// TwinCAT 3 PLC project lev_fsm
// ProgramVersion: 3.1.4023.0
// libraries:
//   Tc2_SerialCom, * (Beckhoff Automation GmbH)
//   Tc2_Standard, * (Beckhoff Automation GmbH)
//   Tc2_System, * (Beckhoff Automation GmbH)
//   Tc2_Utilities, * (Beckhoff Automation GmbH)
//   Tc3_Module, * (Beckhoff Automation GmbH)
// project tree:
//   DUTs/ E_FsmError.TcDUT, E_FsmState.TcDUT, mag_bus.TcDUT, ST_Event.TcDUT, sus_bus.TcDUT
//   / PlcTask.TcTTO
//   POUs/ getTrajectory.TcPOU (not stored), LevitationEqualizingController.TcPOU, MAIN.TcPOU, runIpcFsm.TcPOU (not stored)
//   POUs/outdated/ FiniteStateMachine.TcPOU (not stored), GenerateTrajectory.TcPOU, getFmagnetic.TcPOU, Trajectory.TcPOU (not stored), UpdateEventTimestampWithSystemTime.TcPOU (not stored)

CONFIGURATION lev_fsm
    RESOURCE PLC ON TwinCAT3
        TASK PlcTask(INTERVAL := T#10ms, PRIORITY := 6);
        PROGRAM MAIN WITH PlcTask : MAIN;
    END_RESOURCE
END_CONFIGURATION

// ---- DUTs/E_FsmError.TcDUT
{attribute 'qualified_only'}
{attribute 'strict'}
{attribute 'to_string'}
TYPE E_FsmError :
(
	NO_ERR		  := 0,
	INIT_ERR      := 1,
	STAT_ERR      := 2,
	STAT_TR_ERR   := 3,
	NOM_LEV_ERR   := 4,
	INTER_TR_ERR  := 5,
	END_TR_ERR    := 6
);
END_TYPE

// ---- DUTs/E_FsmState.TcDUT
{attribute 'qualified_only'}
{attribute 'strict'}
{attribute 'to_string'}
TYPE E_FsmState :
(
	ERR       := 0,
	INIT      := 1,
	STAT      := 2, 
	STAT_TR   := 3,
	NOM_LEV   := 4,
	INTER_TR  := 5,
	END_TR 	  := 6
);
END_TYPE

// ---- DUTs/mag_bus.TcDUT
TYPE mag_bus:
    STRUCT
        Fmat: ARRAY [0..143] OF LREAL;
        zmat: ARRAY [0..143] OF LREAL;
        invFmat: ARRAY [0..143] OF LREAL;
        F_grid: ARRAY [0..16383] OF LREAL;
        z_grid: ARRAY [0..16383] OF LREAL;
        i_grid: ARRAY [0..16383] OF LREAL;
    END_STRUCT
END_TYPE

// ---- DUTs/ST_Event.TcDUT
TYPE ST_Event :
STRUCT
	eEventType : E_TcEventClass;
	eEventSeverity : TcEventSeverity;
	nEventID : UDINT;
	sEventDescription : STRING(255);
	dtTimestamp : DATE_AND_TIME;
END_STRUCT
END_TYPE

// ---- DUTs/sus_bus.TcDUT
TYPE sus_bus:
    STRUCT
        zmax: LREAL;
        zcont: LREAL;
    END_STRUCT
END_TYPE

// ---- POUs/MAIN.TcPOU
PROGRAM MAIN

VAR CONSTANT
	tTIMER_TRESHOLD: TIME := T#10S;
END_VAR

VAR
	// LOGGING 
	fbOpenLogFile : FB_FileOpen := (sPathName:='.\logs\ipc.log', nMode:= FOPEN_MODEAPPEND OR FOPEN_MODETEXT);
    fbPutsLogFile : FB_FilePuts;		
	// Reference vector
	x_ref : ARRAY[1..3] OF REAL := [0.01, 0, 32.5]; // [z_nom, v_des, I_nom]
	z_nom : REAL := x_ref[1]; // Nominal air gap
	v_des : REAL := x_ref[2]; // Desired vertical velocity at nominal state
	I_nom: REAL := x_ref[3]; // Nominal current	
	eFsmState : E_FsmState := E_FsmState.INIT; // Finite State Machine State initialization
	eNextFsmState : E_FsmState := E_FsmState.INIT; // Next Finite State Machine State initialization
	stEvent : ST_Event; // Finite State Machine Event definition
	eFsmErrorStatus : E_FsmError; // Finite State Machine Error status
	
	fbTimer: TON := (PT:= tTIMER_TRESHOLD);
	bTimerStart: BOOL := TRUE;
	
	pz_nom : POINTER TO REAL := ADR(z_nom);
	rz_nom : REFERENCE TO REAL REF=z_nom;
	bRunOnlyOnce: BOOL := FALSE;
	nSizeOfLoggerMessage: UINT;
	sLoggerMessage: STRING(100) := 'Logging Finite State Machine State';
	tTime: TIME := T#0D0H0M0S0MS;
	
	// Levitation Equalizing Controller
	fSetpointValue : LREAL := 0; // Reference delta F = 0 N
	bReset : BOOL; // Reset flag for PID block
	fCtrlCycleTime : LREAL := 0.1; // Update cycle time of PID block
	fKp : LREAL := 1/1000;  // Proportional gain of PID block
	fTn : LREAL := 1/150; 
	fTv : LREAL := 0;
	fTd : LREAL := 0;
	fCtrlOutput : LREAL; // Output of PID block
	nErrorStatus : UINT; // Error status of levitation equalizing controller
	// Levitation equalizing controller function block initialization
	LevEqCtrl : LevitationEqualizingController(fSetpointValue := fSetpointValue,
											   bReset := bReset,
                                               fCtrlCycleTime := fCtrlCycleTime,
											   fKp := fKp,
											   fTn := fTn,
											   fTv := fTv,
											   fTd := fTd);
	fActualdF : LREAL; // Actual delta F = (F1 + F3) - (F2 + F4)
	fdz : ARRAY[1..4] OF LREAL;	// dz output vector of levitation equalizing controller
	// Forces
	fFmagFL : LREAL;
	fFmagFR : LREAL;
	fFmagBR : LREAL;
	fFmagBL : LREAL;
	// Test current, airgap and magnetic force
	fztest : LREAL;
	fItest : LREAL;
	fFmagtest : LREAL;
END_VAR

eFsmErrorStatus := runIpcFsm(eFsmState, eNextFsmState, fbTimer, bTimerStart);
fActualdF := (fFmagFL + fFmagBR) - (fFmagFR + fFmagBL);
LevEqCtrl(fActualdF := fActualdF, fdz => fdz, nErrorStatus => nErrorStatus);

fFmagtest := getFmagnetic(fItest,fztest);





(*
IF NOT bRunOnlyOnce THEN
	eNextFsmState := FiniteStateMachine(eArgFsmState := eFsmState);
	pz_nom^ := 0.015;
	x_ref := GenerateTrajectory(z_meas := 0.015, v_meas := 0.01, I_meas := 40);
	stEvent.sEventDescription := 'Start magnetic suspension';
	UpdateEventTimestampWithSystemTime(stEvent := stEvent);
	nSizeOfLoggerMessage := SIZEOF(sLoggerMessage);
	ADSLOGSTR(msgCtrlMask := ADSLOG_MSGTYPE_ERROR OR ADSLOG_MSGTYPE_LOG, 
		  msgFmtStr := sLoggerMessage,
		  strArg := '');
	bRunOnlyOnce := TRUE;
END_IF	 
*)

END_PROGRAM

// ---- POUs/LevitationEqualizingController.TcPOU
FUNCTION_BLOCK LevitationEqualizingController
VAR_INPUT
	// Actual delta F value
	fActualdF : LREAL;
END_VAR

VAR
	// PID function block	
	fbPID : FB_BasicPID;
	// PID parameters
	fSetpointValue : LREAL;
	bReset : BOOL;
	fCtrlCycleTime : LREAL;
	fKp : LREAL;
	fTn : LREAL;
	fTv : LREAL;
	fTd : LREAL;
	// PID outputs	
	fCtrlOutput : LREAL;
	// Saturation parameter
	fdzMax : LREAL := 0.001;
	fdzMin : LREAL := -0.001;
END_VAR
VAR_OUTPUT
	// dz output vector
	fdz : ARRAY[1..4] OF LREAL;
	nErrorStatus : UINT;
END_VAR

fbPID(fSetpointValue := fSetpointValue,
	  fActualValue := fActualdF,
	  bReset := bReset,
	  fCtrlCycleTime := fCtrlCycleTime,
	  fKp := fKp,
	  fTn := fTn,
	  fTv := fTv,
	  fTd := fTd,
	  fCtrlOutput => fCtrlOutput, nErrorStatus => nErrorStatus);
	  
// Update the dz output vector
fdz[1] := -1/7900*fCtrlOutput; // TO DO : change it to lookup table function F_inv(F)
fdz[2] := 1/7900*fCtrlOutput;
fdz[3] := -1/7900*fCtrlOutput;
fdz[4] := 1/7900*fCtrlOutput;	  

// Saturate the dz output vector
IF fdz[1] > fdzMax THEN
	fdz[1] := fdzMax;
ELSIF fdz[1] < fdzMin THEN
	fdz[1] := fdzMin;
END_IF

IF fdz[2] > fdzMax THEN
	fdz[2] := fdzMax;
ELSIF fdz[2] < fdzMin THEN
	fdz[2] := fdzMin;
END_IF

IF fdz[3] > fdzMax THEN
	fdz[3] := fdzMax;
ELSIF fdz[3] < fdzMin THEN
	fdz[3] := fdzMin;
END_IF

IF fdz[4] > fdzMax THEN
	fdz[4] := fdzMax;
ELSIF fdz[4] < fdzMin THEN
	fdz[4] := fdzMin;
END_IF

METHOD FB_init : BOOL
VAR_INPUT
	bInitRetains : BOOL; // if TRUE, the retain variables are initialized (warm start / cold start)
	bInCopyCode : BOOL;  // if TRUE, the instance afterwards gets moved into the copy code (online change)
	fSetpointValue : LREAL;
	bReset : BOOL;
	fCtrlCycleTime : LREAL;
	fKp : LREAL;
	fTn : LREAL;
	fTv : LREAL;
	fTd : LREAL;
END_VAR
THIS^.fSetpointValue := fSetpointValue;
THIS^.bReset := bReset;
THIS^.fCtrlCycleTime := fCtrlCycleTime;
THIS^.fKp := fKp;
THIS^.fTn := fTn;
THIS^.fTv := fTv;
THIS^.fTd := fTd;
END_METHOD

END_FUNCTION_BLOCK

// ---- POUs/outdated/getFmagnetic.TcPOU
FUNCTION getFmagnetic : LREAL
VAR_INPUT
    I: LREAL;
    z: LREAL;
END_VAR
VAR
    Fmag_tmp: LREAL;
    Fmag_tmp_0: LREAL;
    Fmag_tmp_1: LREAL;
    Fmag_tmp_2: LREAL;
    Fmag_tmp_3: LREAL;
    Fmag_tmp_4: LREAL;
END_VAR

(* MATLAB Function: '<Root>/getFmag' *)
(* MATLAB Function 'getFmag': '<S1>:1' *)
(* '<S1>:1:2' p00 =  -4.108e+05; *)
(* '<S1>:1:3' p10 =        3267; *)
(* '<S1>:1:4' p01 =   1.697e+05; *)
(* '<S1>:1:5' p20 =       61.45; *)
(* '<S1>:1:6' p11 =       -1147; *)
(* '<S1>:1:7' p02 =   -2.79e+04; *)
(* '<S1>:1:8' p30 =     -0.5002; *)
(* '<S1>:1:9' p21 =      -8.054; *)
(* '<S1>:1:10' p12 =       147.8; *)
(* '<S1>:1:11' p03 =        2282; *)
(* '<S1>:1:12' p40 =    -0.01962; *)
(* '<S1>:1:13' p31 =      0.1688; *)
(* '<S1>:1:14' p22 =      0.1559; *)
(* '<S1>:1:15' p13 =      -8.184; *)
(* '<S1>:1:16' p04 =      -92.92; *)
(* '<S1>:1:17' p50 =   0.0002649; *)
(* '<S1>:1:18' p41 =   -0.001089; *)
(* '<S1>:1:19' p32 =   -0.001289; *)
(* '<S1>:1:20' p23 =   -0.003046; *)
(* '<S1>:1:21' p14 =      0.1725; *)
(* '<S1>:1:22' p05 =       1.506; *)
(* '<S1>:1:23' Fmag = p00 + p10*I + p01*z + p20*I^2 + p11*I*z + p02*z^2 + p30*I^3 + p21*I^2*z + p12*I*z^2 + p03*z^3 + p40*I^4 + p31*I^3*z + p22*I^2*z^2 + p13*I*z^3 + p04*z^4 + p50*I^5 + p41*I^4*z + p32*I^3*z^2 + p23*I^2*z^3 + p14*I*z^4 + p05*z^5; *)
Fmag_tmp := EXPT(I, 3.0);
Fmag_tmp_0 := EXPT(z, 3.0);
Fmag_tmp_1 := EXPT(I, 4.0);
Fmag_tmp_2 := EXPT(z, 4.0);
Fmag_tmp_3 := I * I;
Fmag_tmp_4 := z * z;
getFmagnetic := ((((((((((((((((((((3267.0 * I) - 410800.0) + (169700.0 * z)) + (Fmag_tmp_3 * 61.45)) + ((-1147.0 * I) * z)) + (Fmag_tmp_4 * -27900.0)) + (-0.5002 * Fmag_tmp)) + ((Fmag_tmp_3 * -8.054) * z)) + ((147.8 * I) * Fmag_tmp_4)) + (2282.0 * Fmag_tmp_0)) + (-0.01962 * Fmag_tmp_1)) + ((0.1688 * Fmag_tmp) * z)) + ((Fmag_tmp_3 * 0.1559) * Fmag_tmp_4)) + ((-8.184 * I) * Fmag_tmp_0)) + (-92.92 * Fmag_tmp_2)) + (0.0002649 * EXPT(I, 5.0))) + ((-0.001089 * Fmag_tmp_1) * z)) + ((-0.001289 * Fmag_tmp) * Fmag_tmp_4)) + ((Fmag_tmp_3 * -0.003046) * Fmag_tmp_0)) + ((0.1725 * I) * Fmag_tmp_2)) + (1.506 * EXPT(z, 5.0));

END_FUNCTION

// ---- POUs/outdated/GenerateTrajectory.TcPOU
(*FUNCTION GenerateTrajectory :  ARRAY[1..3] OF REAL
VAR_INPUT
	z_meas : REAL;
	v_meas : REAL;
	I_meas : REAL;
END_VAR
VAR
END_VAR*)
(*
 *
 * File: trajectory_generator.st
 *
 * IEC 61131-3 Structured Text (ST) code generated for subsystem "trajectory_generator/getTrajectory"
 *
 * Model name                      : trajectory_generator
 * Model version                   : 3.24
 * Model creator                   : xiaomi
 * Model last modified by          : xiaomi
 * Model last modified on          : Tue Oct 25 16:42:44 2022
 * Model sample time               : 0.0005s
 * Subsystem name                  : trajectory_generator/getTrajectory
 * Subsystem sample time           : 0.1s
 * Simulink PLC Coder version      : 3.7 (R2022b) 13-May-2022
 * ST code generated on            : Tue Oct 25 16:44:27 2022
 *
 * Target IDE selection            : Beckhoff TwinCAT 3
 * Test Bench included             : No
 *
 *)
FUNCTION_BLOCK GenerateTrajectory
VAR_INPUT
    ssMethodType: SINT;
    t: LREAL;
    Tdes: LREAL;
    z0: LREAL;
    v0: LREAL;
    a0: LREAL;
    zdes: LREAL;
    vdes: LREAL;
    ades: LREAL;
    sus_params: sus_bus;
    mag_params: mag_bus;
END_VAR
VAR_OUTPUT
    zd: LREAL;
    vd: LREAL;
    ad: LREAL;
    id: LREAL;
END_VAR
VAR
    zd_prev_not_empty: BOOL;
    zd_prev: LREAL;
    vd_prev_not_empty: BOOL;
    vd_prev: LREAL;
    ad_prev_not_empty: BOOL;
    ad_prev: LREAL;
    id_prev: LREAL;
END_VAR
VAR_TEMP
    b2: LREAL;
    Fsus: LREAL;
    K: LREAL;
    zd_norm: LREAL;
    Fmag_norm: LREAL;
    A: ARRAY [0..8] OF LREAL;
    B: ARRAY [0..2] OF LREAL;
    r1: DINT;
    r2: DINT;
    r3: DINT;
    maxval: LREAL;
    a21: LREAL;
    rtemp: DINT;
    v: ARRAY [0..29] OF LREAL;
    b_v: ARRAY [0..15] OF LREAL;
    ry: LREAL;
    b_mid_i: DINT;
    x_idx_1: LREAL;
    x_idx_2: LREAL;
    x_idx_0: LREAL;
    u: DINT;
    b_u: DINT;
END_VAR

VAR CONSTANT
    SS_INITIALIZE: SINT := 0;
    SS_STEP: SINT := 1;
END_VAR

(*GenerateTrajectory[1] := z_meas/2;
GenerateTrajectory[2] := 0;
GenerateTrajectory[3] := I_meas/2;*)
CASE ssMethodType OF
    SS_INITIALIZE: 
        (* SystemInitialize for MATLAB Function: '<Root>/getTrajectory' *)
        zd_prev_not_empty := FALSE;
        vd_prev_not_empty := FALSE;
        ad_prev_not_empty := FALSE;
        (* '<S1>:1:25' id_prev = 0; *)
        id_prev := 0.0;
    SS_STEP: 
        (* MATLAB Function: '<Root>/getTrajectory' *)
        (* %% Solve the system of equations *)
        (* MATLAB Function 'getTrajectory': '<S1>:1' *)
        (* '<S1>:1:4' T_matrix = [ Tdes^3 Tdes^4 Tdes^5; 3*Tdes^2 4*Tdes^3 5*Tdes^4; 6*Tdes 12*Tdes^2 20*Tdes^3]; *)
        maxval := EXPT(Tdes, 3.0);
        a21 := EXPT(Tdes, 4.0);
        (* MATLAB Function: '<Root>/getTrajectory' incorporates:
         *  Inport: '<Root>/mag_params' *)
        A[0] := maxval;
        A[3] := a21;
        A[6] := EXPT(Tdes, 5.0);
        ry := Tdes * Tdes;
        A[1] := ry * 3.0;
        A[4] := 4.0 * maxval;
        A[7] := 5.0 * a21;
        A[2] := 6.0 * Tdes;
        A[5] := ry * 12.0;
        A[8] := 20.0 * maxval;
        (* '<S1>:1:5' y = [zdes-z0-v0*Tdes-a0/2*Tdes^2; vdes-v0-a0*Tdes; ades-a0]; *)
        B[0] := ((zdes - z0) - (v0 * Tdes)) - ((a0 / 2.0) * ry);
        B[1] := (vdes - v0) - (a0 * Tdes);
        B[2] := ades - a0;
        (* '<S1>:1:6' x = T_matrix\y; *)
        r1 := 0;
        r2 := 1;
        r3 := 2;
        maxval := ABS(maxval);
        a21 := ABS(A[1]);
        IF a21 > maxval THEN 
            maxval := a21;
            r1 := 1;
            r2 := 0;
        END_IF;
        IF ABS(A[2]) > maxval THEN 
            r1 := 2;
            r2 := 1;
            r3 := 0;
        END_IF;
        A[r2] := A[r2] / A[r1];
        A[r3] := A[r3] / A[r1];
        A[r2 + 3] := A[r2 + 3] - (A[r1 + 3] * A[r2]);
        A[r3 + 3] := A[r3 + 3] - (A[r1 + 3] * A[r3]);
        A[r2 + 6] := A[r2 + 6] - (A[r1 + 6] * A[r2]);
        A[r3 + 6] := A[r3 + 6] - (A[r1 + 6] * A[r3]);
        IF ABS(A[r3 + 3]) > ABS(A[r2 + 3]) THEN 
            rtemp := r2;
            r2 := r3;
            r3 := rtemp;
        END_IF;
        A[r3 + 3] := A[r3 + 3] / A[r2 + 3];
        A[r3 + 6] := A[r3 + 6] - (A[r3 + 3] * A[r2 + 6]);
        x_idx_1 := B[r2] - (B[r1] * A[r2]);
        x_idx_2 := ((B[r3] - (B[r1] * A[r3])) - (A[r3 + 3] * x_idx_1)) / A[r3 + 6];
        x_idx_1 := (x_idx_1 - (A[r2 + 6] * x_idx_2)) / A[r2 + 3];
        x_idx_0 := ((B[r1] - (A[r1 + 6] * x_idx_2)) - (A[r1 + 3] * x_idx_1)) / A[r1];
        (* %% Define the trajectory polynomial coefficiets *)
        (* '<S1>:1:8' b0 = z0; *)
        (* '<S1>:1:9' b1 = v0; *)
        (* '<S1>:1:10' b2 = a0/2; *)
        b2 := a0 / 2.0;
        (* '<S1>:1:11' b3 = x(1); *)
        (* '<S1>:1:12' b4 = x(2); *)
        (* '<S1>:1:13' b5 = x(3); *)
        (* '<S1>:1:15' if isempty(zd_prev) *)
        IF  NOT zd_prev_not_empty THEN 
            (* '<S1>:1:16' zd_prev = z0; *)
            zd_prev := z0;
            zd_prev_not_empty := TRUE;
        END_IF;
        (* '<S1>:1:18' if isempty(vd_prev) *)
        IF  NOT vd_prev_not_empty THEN 
            (* '<S1>:1:19' vd_prev = v0; *)
            vd_prev := v0;
            vd_prev_not_empty := TRUE;
        END_IF;
        (* '<S1>:1:21' if isempty(ad_prev) *)
        IF  NOT ad_prev_not_empty THEN 
            (* '<S1>:1:22' ad_prev = a0; *)
            ad_prev := a0;
            ad_prev_not_empty := TRUE;
        END_IF;
        (* '<S1>:1:24' if isempty(id_prev) *)
        (* '<S1>:1:27' if t <= Tdes *)
        IF t <= Tdes THEN 
            (* %% Define the trajectory polynomial functions *)
            (* '<S1>:1:29' zd = b0 + b1*t + b2*t^2 + b3*t^3 + b4*t^4 + b5*t^5; *)
            maxval := EXPT(t, 3.0);
            a21 := EXPT(t, 4.0);
            ry := t * t;
            zd := (((((v0 * t) + z0) + (ry * b2)) + (x_idx_0 * maxval)) + (x_idx_1 * a21)) + (x_idx_2 * EXPT(t, 5.0));
            (* '<S1>:1:30' vd = b1 + 2*b2*t + 3*b3*t^2 + 4*b4*t^3 + 5*b5*t^4; *)
            vd := (((((2.0 * b2) * t) + v0) + ((3.0 * x_idx_0) * ry)) + ((4.0 * x_idx_1) * maxval)) + ((5.0 * x_idx_2) * a21);
            (* '<S1>:1:31' ad = 2*b2 + 6*b3*t + 12*b4*t^2 + 20*b5*t^3; *)
            ad := ((((6.0 * x_idx_0) * t) + (2.0 * b2)) + ((12.0 * x_idx_1) * ry)) + ((20.0 * x_idx_2) * maxval);
            (* %% Find id through system dynamics model *)
            (* '<S1>:1:34' M = 1000; *)
            (* mass  *)
            (* '<S1>:1:35' g = 9.81; *)
            (* gravitational acceleration *)
            (* '<S1>:1:36' Fres = ad*M; *)
            (* resultant force *)
            (* '<S1>:1:37' Fg = g*M; *)
            (* gravitational force *)
            (* '<S1>:1:38' Fsus = susModel(zd,sus_params,Fg); *)
            (* 'susModel:2' zmax = sus_params.zmax; *)
            (* 'susModel:3' zcont = sus_params.zcont; *)
            (* 'susModel:4' Fmax = Fg; *)
            (* 'susModel:5' Fmin = 0; *)
            (* 'susModel:7' K = (Fmax - Fmin) / (zmax - zcont); *)
            K := 9810.0 / (sus_params.zmax - sus_params.zcont);
            (* 'susModel:8' N = Fmax - K * zmax; *)
            (* 'susModel:10' if zd > zmax *)
            IF zd > sus_params.zmax THEN 
                (* 'susModel:11' Fsus = Fg; *)
                Fsus := 9810.0;
            ELSIF zd < sus_params.zcont THEN 
                (* 'susModel:12' elseif zd < zcont *)
                (* 'susModel:13' Fsus = 0; *)
                Fsus := 0.0;
            ELSE 
                (* 'susModel:14' else *)
                (* 'susModel:15' Fsus = K * zd + N; *)
                Fsus := (9810.0 - (K * sus_params.zmax)) + (K * zd);
            END_IF;
            (* suspenssion force *)
            (* '<S1>:1:39' Fmag = Fg - Fsus - Fres; *)
            (* magnetic force (second newton law) *)
            (* use the inverse force model to compute the desired current for the specified force and distance *)
            (* '<S1>:1:41' id = invForceModel(Fmag,zd,mag_params); *)
            (* %% parameters *)
            (* 'invForceModel:3' znorm = mag_params.znorm; *)
            (* normalising constant for the input distance (1/zmax) *)
            (* 'invForceModel:4' Fnorm = mag_params.Fnorm; *)
            (* normalising constant for the input force (1/Fmax) *)
            (* 'invForceModel:5' invFmax =  mag_params.invFmax; *)
            (* gain for the inverse matrix (this is actually Imax) *)
            (* 'invForceModel:6' zmat = mag_params.zmat; *)
            (* (input) distance matrix  *)
            (* 'invForceModel:7' Fmat = mag_params.Fmat; *)
            (* (input) force matrix  *)
            (* 'invForceModel:8' invFmat = mag_params.invFmat; *)
            (* (output) inverse force matrix - this is actually a current matrix  *)
            (* 'invForceModel:11' zd_norm = zd * znorm; *)
            zd_norm := zd * mag_params.znorm;
            (* normalised input distance     *)
            (* 'invForceModel:12' Fmag_norm = Fmag * Fnorm; *)
            Fmag_norm := ((9810.0 - Fsus) - (ad * 1000.0)) * mag_params.Fnorm;
            (* normalised input force *)
            (* %% compute desired current *)
            (* 'invForceModel:16' if (Fmag_norm > 1) *)
            IF Fmag_norm > 1.0 THEN 
                (* force is out of range *)
                (* 'invForceModel:17' id = invFmax; *)
                id := mag_params.invFmax;
            ELSIF Fmag_norm < 0.0 THEN 
                (* 'invForceModel:18' elseif (Fmag_norm <0) *)
                (* force is smaller than zero *)
                (* 'invForceModel:19' id = 0; *)
                id := 0.0;
            ELSE 
                (* 'invForceModel:20' else *)
                (* 'invForceModel:21' id = invFmax * interp2(Fmat, zmat, invFmat, Fmag_norm, zd_norm); *)
                FOR r1 := 0 TO 29 DO 
                    v[r1] := mag_params.Fmat[r1 * 16];
                END_FOR;
                FOR r1 := 0 TO 15 DO 
                    b_v[r1] := mag_params.zmat[r1];
                END_FOR;
                IF Fmag_norm >= v[0] THEN 
                    IF Fmag_norm <= v[29] THEN 
                        IF zd_norm >= b_v[0] THEN 
                            IF zd_norm <= b_v[15] THEN 
                                r2 := 30;
                                r1 := 0;
                                r3 := 2;
                                WHILE r2 > r3 DO
                                    u := (r1 + r2) + 1;
                                    IF u >= 0 THEN 
                                        rtemp := UDINT_TO_DINT(DWORD_TO_UDINT(SHR(UDINT_TO_DWORD(DINT_TO_UDINT(u)), 1)));
                                    ELSE 
                                        rtemp := ( -UDINT_TO_DINT(DWORD_TO_UDINT(SHR(UDINT_TO_DWORD(DINT_TO_UDINT(-1 - u)), 1)))) - 1;
                                    END_IF;
                                    IF Fmag_norm >= v[rtemp - 1] THEN 
                                        r1 := rtemp - 1;
                                        r3 := rtemp + 1;
                                    ELSE 
                                        r2 := rtemp;
                                    END_IF;
                                END_WHILE;
                                r2 := 16;
                                r3 := 1;
                                rtemp := 2;
                                WHILE r2 > rtemp DO
                                    b_u := r3 + r2;
                                    IF b_u >= 0 THEN 
                                        b_mid_i := UDINT_TO_DINT(DWORD_TO_UDINT(SHR(UDINT_TO_DWORD(DINT_TO_UDINT(b_u)), 1)));
                                    ELSE 
                                        b_mid_i := ( -UDINT_TO_DINT(DWORD_TO_UDINT(SHR(UDINT_TO_DWORD(DINT_TO_UDINT(-1 - b_u)), 1)))) - 1;
                                    END_IF;
                                    IF zd_norm >= b_v[b_mid_i - 1] THEN 
                                        r3 := b_mid_i;
                                        rtemp := b_mid_i + 1;
                                    ELSE 
                                        r2 := b_mid_i;
                                    END_IF;
                                END_WHILE;
                                IF Fmag_norm = v[r1] THEN 
                                    r1 := DWORD_TO_DINT(SHL(DINT_TO_DWORD(r1), 4)) + r3;
                                    maxval := mag_params.invFmat[r1 - 1];
                                    a21 := mag_params.invFmat[r1];
                                ELSE 
                                    ry := v[r1 + 1];
                                    IF ry = Fmag_norm THEN 
                                        r1 := DWORD_TO_DINT(SHL(DINT_TO_DWORD(r1 + 1), 4)) + r3;
                                        maxval := mag_params.invFmat[r1 - 1];
                                        a21 := mag_params.invFmat[r1];
                                    ELSE 
                                        a21 := (Fmag_norm - v[r1]) / (ry - v[r1]);
                                        ry := mag_params.invFmat[(((r1 + 1) * 16) + r3) - 1];
                                        r2 := (DWORD_TO_DINT(SHL(DINT_TO_DWORD(r1), 4)) + r3) - 1;
                                        maxval := mag_params.invFmat[r2];
                                        IF ry = maxval THEN 
                                            maxval := mag_params.invFmat[r2];
                                        ELSE 
                                            maxval := (ry * a21) + (maxval * (1.0 - a21));
                                        END_IF;
                                        r2 := DWORD_TO_DINT(SHL(DINT_TO_DWORD(r1 + 1), 4)) + r3;
                                        r1 := DWORD_TO_DINT(SHL(DINT_TO_DWORD(r1), 4)) + r3;
                                        IF mag_params.invFmat[r2] = mag_params.invFmat[r1] THEN 
                                            a21 := mag_params.invFmat[r1];
                                        ELSE 
                                            a21 := (mag_params.invFmat[r2] * a21) + (mag_params.invFmat[r1] * (1.0 - a21));
                                        END_IF;
                                    END_IF;
                                END_IF;
                                ry := b_v[r3 - 1];
                                IF ry = zd_norm THEN 
                                    a21 := maxval;
                                ELSIF maxval = a21 THEN 
                                    a21 := maxval;
                                ELSIF zd_norm <> b_v[r3] THEN 
                                    ry := (zd_norm - ry) / (b_v[r3] - ry);
                                    a21 := ((1.0 - ry) * maxval) + (ry * a21);
                                END_IF;
                            ELSE 
                                a21 := 0.0;
                            END_IF;
                        ELSE 
                            a21 := 0.0;
                        END_IF;
                    ELSE 
                        a21 := 0.0;
                    END_IF;
                ELSE 
                    a21 := 0.0;
                END_IF;
                id := mag_params.invFmax * a21;
            END_IF;
            (* %% Update previous values *)
            (* '<S1>:1:44' zd_prev = zd; *)
            zd_prev := zd;
            (* '<S1>:1:45' vd_prev = vd; *)
            vd_prev := vd;
            (* '<S1>:1:46' ad_prev = ad; *)
            ad_prev := ad;
            (* '<S1>:1:47' id_prev = id; *)
            id_prev := id;
        ELSE 
            (* '<S1>:1:48' else *)
            (* %% Keep previous values *)
            (* '<S1>:1:50' zd = zd_prev; *)
            zd := zd_prev;
            (* '<S1>:1:51' vd = vd_prev; *)
            vd := vd_prev;
            (* '<S1>:1:52' ad = ad_prev; *)
            ad := ad_prev;
            (* '<S1>:1:53' id = id_prev; *)
            id := id_prev;
        END_IF;
END_CASE;

END_FUNCTION_BLOCK
